{attribute 'linkalways'} 
{attribute 'no_explicit_call' := 'This FB is a CLASS and must be accessed using methods or properties'}
{attribute 'enable_dynamic_creation'}
FUNCTION_BLOCK Node_F_VN_CompensateLensDistortionForPointsExp2 EXTENDS VisionNode
VAR
    ipSrcPoints : _ITcVnContainer;
    ipDestPoints : _ITcVnContainer;
    aCameraMatrix : _TcVnMatrix3x3_LREAL;
    aDistortionCoefficients : _TcVnArray8_LREAL;
    aNewCameraMatrix : _TcVnMatrix3x3_LREAL;
    hrPrev : _HRESULT(S_OK);
	hresult : _HRESULT(S_OK);
END_VAR

METHOD PUBLIC  Clone : I_Node
VAR
	pNode : POINTER TO Node_F_VN_CompensateLensDistortionForPointsExp2;
END_VAR
pNode := __NEW(Node_F_VN_CompensateLensDistortionForPointsExp2);
Clone := pNode^;
END_METHOD

METHOD FB_init : BOOL
VAR_INPUT
	bInitRetains : BOOL; // if TRUE, the retain variables are initialized (warm start / cold start)
	bInCopyCode : BOOL;  // if TRUE, the instance afterwards gets moved into the copy code (online change)
END_VAR
AddInput('ipSrcPoints', ipSrcPoints);
AddInput('aCameraMatrix', aCameraMatrix);
AddInput('aDistortionCoefficients', aDistortionCoefficients);
AddInput('aNewCameraMatrix', aNewCameraMatrix);
AddInput('hrPrev', hrPrev);
AddOutput('ipDestPoints', ipDestPoints);
AddOutput('hresult', hresult);
END_METHOD

METHOD PROTECTED OnExecute
hresult.Value := F_VN_CompensateLensDistortionForPointsExp2(
    ipSrcPoints := ipSrcPoints.Value,
	ipDestPoints := ipDestPoints.Value,
    aCameraMatrix := aCameraMatrix.Value,
    aDistortionCoefficients := aDistortionCoefficients.Value,
    aNewCameraMatrix := aNewCameraMatrix.Value,
	hrPrev := hrPrev.Value);
END_METHOD

METHOD PUBLIC PreExecutionCheck
VAR_INPUT
	Check : I_PreExecutionChecks;
END_VAR
Check.IsTrue(ipSrcPoints.IsValid, 'ipSrcPoints must be a valid container');
Check.IsTrue((ipSrcPoints.IsType(TC_GLOBAL_CONST_LIST.ContainerType_Vector_TcVnPoint2_DINT) OR
              ipSrcPoints.IsType(TC_GLOBAL_CONST_LIST.ContainerType_Vector_TcVnPoint2_REAL)),
              'ipSrcPoints contains incorrect type');
END_METHOD

END_FUNCTION_BLOCK

(* stored: Version 1.1.0.1, ProductVersion 3.1.4026.13
   POU Node_F_VN_CompensateLensDistortionForPointsExp2: Id {2d4005ed-8862-0ae9-0a39-38412e5f9aa3}, SpecialFunc None
   Folder Constructor: Id {28c3a217-c465-0da1-01bf-4fbeb4152b4c}
   Method Clone: Id {34e5db39-c7fc-0966-1545-1398f0f0e260}
   Method FB_init: Id {7766b0c7-cd03-01a5-0e21-ff8ac12234f9}
   Method OnExecute: Id {bccb45ce-8008-0fbe-08b4-14da9668381d}
   Method PreExecutionCheck: Id {79c3e2d8-cd16-0f17-0f97-5c9f8ab69b13} *)
